FUNCTION_BLOCK FB_Incubator EXTENDS FB_Station
VAR
END_VAR

METHOD Hatching : INT
VAR
	stTempUnit				: ST_Unit;
	iTempIndex				: INT;
	iHatchCounter			: INT;
END_VAR
Hatching := 0;
IF iLastIndex > 0 THEN
	FOR iTempIndex := 1 TO iLastIndex BY 1 DO
		stTempUnit := stUnitArr[iTempIndex];
		IF stTempUnit.iProgress < 6 THEN
			stTempUnit.iProgress := stTempUnit.iProgress + 1;
			stUnitArr[iTempIndex] := stTempUnit;
		ELSE
			RemoveUnit(iTempIndex);
			iHatchCounter := iHatchCounter + 1;
		END_IF
	END_FOR
END_IF
Hatching := iHatchCounter;
END_METHOD

END_FUNCTION_BLOCK

(* stored: Version 1.1.0.1, ProductVersion 3.1.4024.12
   POU FB_Incubator: Id {4bbf2477-6dce-43b6-9a38-1df9d00436a5}, SpecialFunc None
   Method Hatching: Id {20cf3caf-be4c-44da-932d-f076630515bb} *)
